{attribute 'qualified_only'}
TYPE E_GBS_States :
(
    Unknown := 0,
    OUT := 1,
    TARGET1a := 2,
    TARGET1b := 3,
    TARGET2a := 4,
    TARGET2b := 5,
    TARGET3a := 6,
    TARGET3b := 7,
    TARGET4 := 8,
    TARGET5 := 9,
    TARGET6 := 10
) UINT;
END_TYPE

(* stored: Version 1.1.0.1
   DUT E_GBS_States: Id {a23f1263-4eb4-41bc-9092-54ae1e43deed} *)
